Yaskawa INFORM job: _DEL24.JBI

/JOB
//NAME _DEL24
//POS
///NPOS 0,0,0,0,0,0
//INST
///DATE 2018/08/28 16:53
///ATTR SC,RW,CJ,MC
NOP
END
